// Mitsubishi GX Works2 project: 2023-06-21 #1 생산자동화기능사 2번   PLC: Q03UDV
// 생산자동화기능사

// global labels: Global1
VAR_GLOBAL
  PB1 AT X0 : BOOL;
  PB2 AT X1 : BOOL;
  정지 AT X2 : BOOL;
  공급후진 AT X3 : BOOL;
  공급전진 AT X4 : BOOL;
  가공후진 AT X5 : BOOL;
  가공전진 AT X6 : BOOL;
  송출후진 AT X7 : BOOL;
  송출전진 AT X8 : BOOL;
  배출후진 AT X9 : BOOL;
  배출전진 AT X0A : BOOL;
  매거진 AT X0B : BOOL;
  금속센서 AT X0F : BOOL;
  PB3 AT X0C : BOOL;
  적색 AT Y20 : BOOL;
  황색 AT Y21 : BOOL;
  녹색 AT Y22 : BOOL;
  공급1 AT Y23 : BOOL;
  공급2 AT Y24 : BOOL;
  가공 AT Y25 : BOOL;
  드릴 AT Y26 : BOOL;
  송출 AT Y27 : BOOL;
  배출 AT Y28 : BOOL;
  컨베이어 AT Y29 : BOOL;
END_VAR

PROGRAM 테스트동작
VAR
  PHASE : INT;
END_VAR
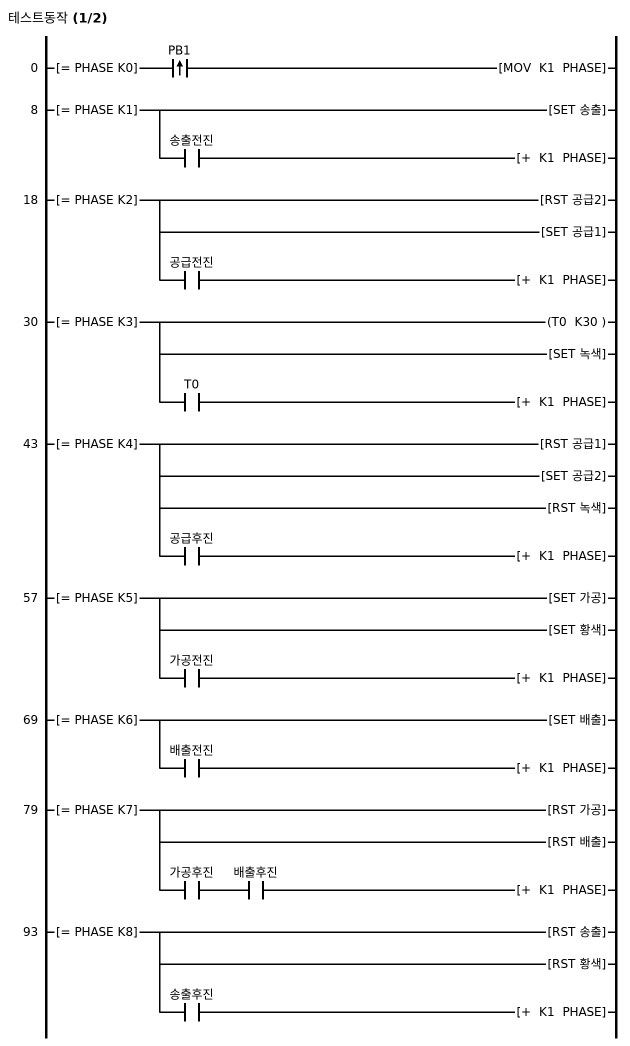
0     LD=     PHASE K0
      ANDP    PB1
      MOV     K1 PHASE
8     LD=     PHASE K1
      SET     송출
      AND     송출전진
      +       K1 PHASE
18    LD=     PHASE K2
      RST     공급2
      SET     공급1
      AND     공급전진
      +       K1 PHASE
30    LD=     PHASE K3
      OUT     T0 K30
      SET     녹색
      AND     T0
      +       K1 PHASE
43    LD=     PHASE K4
      RST     공급1
      SET     공급2
      RST     녹색
      AND     공급후진
      +       K1 PHASE
57    LD=     PHASE K5
      SET     가공
      SET     황색
      AND     가공전진
      +       K1 PHASE
69    LD=     PHASE K6
      SET     배출
      AND     배출전진
      +       K1 PHASE
79    LD=     PHASE K7
      RST     가공
      RST     배출
      AND     가공후진
      AND     배출후진
      +       K1 PHASE
93    LD=     PHASE K8
      RST     송출
      RST     황색
      AND     송출후진
      +       K1 PHASE
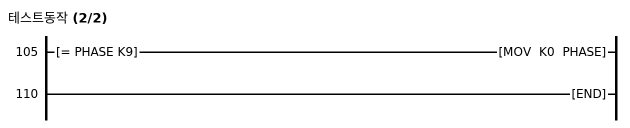
105   LD=     PHASE K9
      MOV     K0 PHASE
110   END
END_PROGRAM

PROGRAM 단속연속동작
VAR
  PHASE : INT;
  MODE : INT;
END_VAR
VAR CONSTANT
  단속 : INT;
  연속 : INT := 1;
END_VAR
VAR
  COUNT : ARRAY [0..0] OF INT;
  EMG : INT;
  BLINK : ARRAY [0..3] OF BOOL;
END_VAR
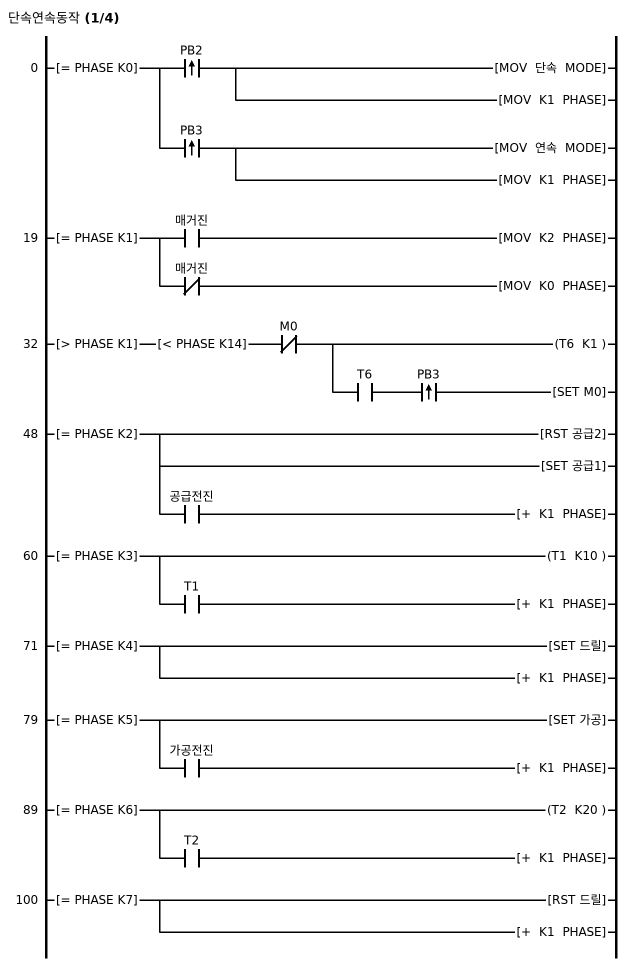
0     LD=     PHASE K0
      MPS
      ANDP    PB2
      MOV     단속 MODE
      MOV     K1 PHASE
      MPP
      ANDP    PB3
      MOV     연속 MODE
      MOV     K1 PHASE
19    LD=     PHASE K1
      MPS
      AND     매거진
      MOV     K2 PHASE
      MPP
      ANI     매거진
      MOV     K0 PHASE
32    LD>     PHASE K1
      AND<    PHASE K14
      ANI     M0
      OUT     T6 K1
      AND     T6
      ANDP    PB3
      SET     M0
48    LD=     PHASE K2
      RST     공급2
      SET     공급1
      AND     공급전진
      +       K1 PHASE
60    LD=     PHASE K3
      OUT     T1 K10
      AND     T1
      +       K1 PHASE
71    LD=     PHASE K4
      SET     드릴
      +       K1 PHASE
79    LD=     PHASE K5
      SET     가공
      AND     가공전진
      +       K1 PHASE
89    LD=     PHASE K6
      OUT     T2 K20
      AND     T2
      +       K1 PHASE
100   LD=     PHASE K7
      RST     드릴
      +       K1 PHASE
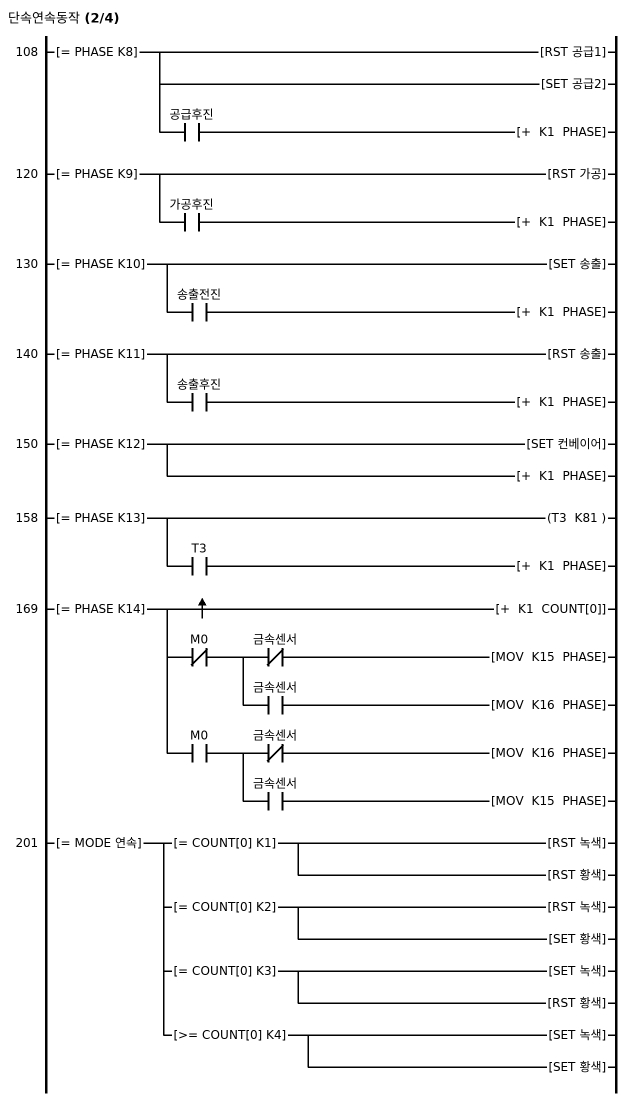
108   LD=     PHASE K8
      RST     공급1
      SET     공급2
      AND     공급후진
      +       K1 PHASE
120   LD=     PHASE K9
      RST     가공
      AND     가공후진
      +       K1 PHASE
130   LD=     PHASE K10
      SET     송출
      AND     송출전진
      +       K1 PHASE
140   LD=     PHASE K11
      RST     송출
      AND     송출후진
      +       K1 PHASE
150   LD=     PHASE K12
      SET     컨베이어
      +       K1 PHASE
158   LD=     PHASE K13
      OUT     T3 K81
      AND     T3
      +       K1 PHASE
169   LD=     PHASE K14
      MPS
      MEP
      +       K1 COUNT[0]
      MRD
      ANI     M0
      MPS
      ANI     금속센서
      MOV     K15 PHASE
      MPP
      AND     금속센서
      MOV     K16 PHASE
      MPP
      AND     M0
      MPS
      ANI     금속센서
      MOV     K16 PHASE
      MPP
      AND     금속센서
      MOV     K15 PHASE
201   LD=     MODE 연속
      MPS
      AND=    COUNT[0] K1
      RST     녹색
      RST     황색
      MRD
      AND=    COUNT[0] K2
      RST     녹색
      SET     황색
      MRD
      AND=    COUNT[0] K3
      SET     녹색
      RST     황색
      MPP
      AND>=   COUNT[0] K4
      SET     녹색
      SET     황색
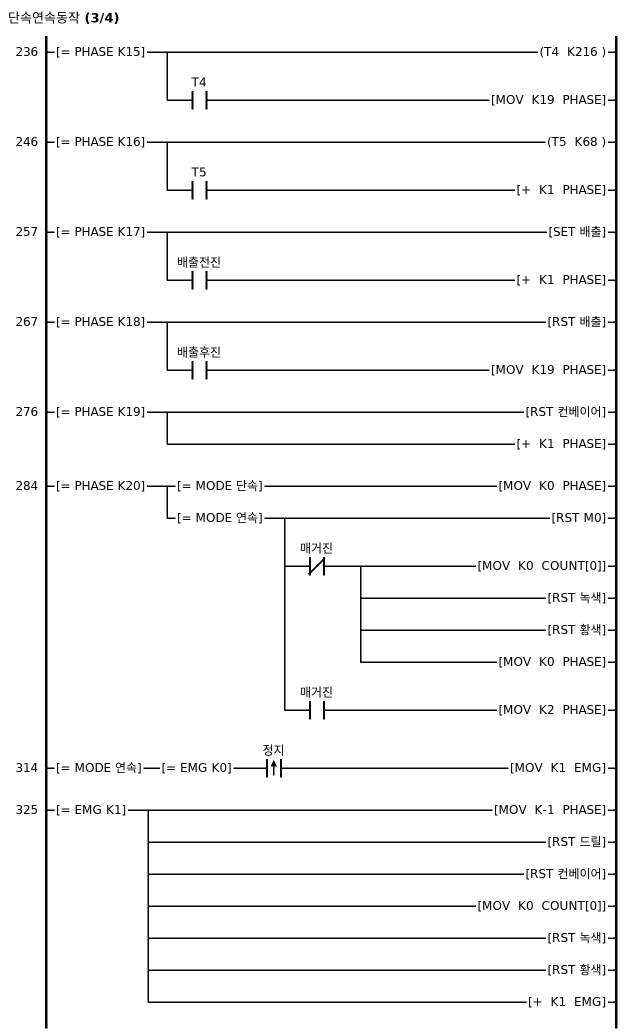
236   LD=     PHASE K15
      OUT     T4 K216
      AND     T4
      MOV     K19 PHASE
246   LD=     PHASE K16
      OUT     T5 K68
      AND     T5
      +       K1 PHASE
257   LD=     PHASE K17
      SET     배출
      AND     배출전진
      +       K1 PHASE
267   LD=     PHASE K18
      RST     배출
      AND     배출후진
      MOV     K19 PHASE
276   LD=     PHASE K19
      RST     컨베이어
      +       K1 PHASE
284   LD=     PHASE K20
      MPS
      AND=    MODE 단속
      MOV     K0 PHASE
      MPP
      AND=    MODE 연속
      RST     M0
      MPS
      ANI     매거진
      MOV     K0 COUNT[0]
      RST     녹색
      RST     황색
      MOV     K0 PHASE
      MPP
      AND     매거진
      MOV     K2 PHASE
314   LD=     MODE 연속
      AND=    EMG K0
      ANDP    정지
      MOV     K1 EMG
325   LD=     EMG K1
      MOV     K-1 PHASE
      RST     드릴
      RST     컨베이어
      MOV     K0 COUNT[0]
      RST     녹색
      RST     황색
      +       K1 EMG
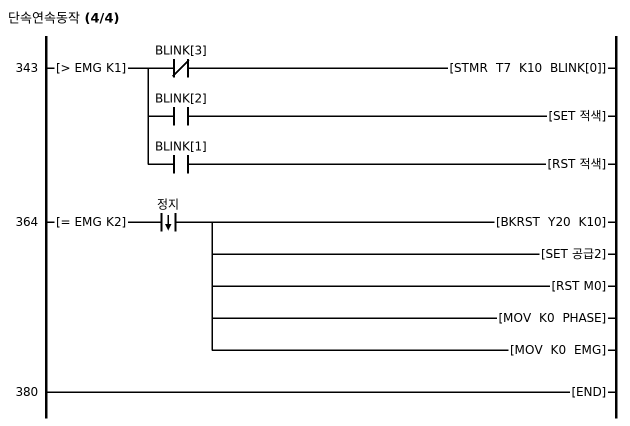
343   LD>     EMG K1
      MPS
      ANI     BLINK[3]
      STMR    T7 K10 BLINK[0]
      MRD
      AND     BLINK[2]
      SET     적색
      MPP
      AND     BLINK[1]
      RST     적색
364   LD=     EMG K2
      ANDF    정지
      BKRST   Y20 K10
      SET     공급2
      RST     M0
      MOV     K0 PHASE
      MOV     K0 EMG
380   END
END_PROGRAM
